// TwinCAT 3 PLC project PLC
// ProgramVersion: 3.1.4023.0
// libraries:
//   Tc2_Standard, * (Beckhoff Automation GmbH)
//   Tc2_System, * (Beckhoff Automation GmbH)
//   Tc3_EventLogger, * (Beckhoff Automation GmbH)
//   Tc3_Module, * (Beckhoff Automation GmbH)
// project tree:
//   GVLs/ GVL.TcGVL
//   / PlcTask.TcTTO
//   POUs/ FB_Alarm.TcPOU, MAIN.TcPOU
// real-time tasks:
//   TASK PlcTask: cycle T#10ms, priority 20, ADS port 350

CONFIGURATION PLC
    RESOURCE PLC ON TwinCAT3
        TASK PlcTask(INTERVAL := T#10ms, PRIORITY := 20);
        PROGRAM MAIN WITH PlcTask : MAIN;
    END_RESOURCE
END_CONFIGURATION

// ---- GVLs/GVL.TcGVL

VAR_GLOBAL

END_VAR

// ---- POUs/MAIN.TcPOU
PROGRAM MAIN
VAR
	// Variables for the FB_TcMessage example
	bInitEvent1 	: BOOL; 
	bInitEvent2 	: BOOL; 
    bSend 			: BOOL; 
	fbMessage 		: FB_TcMessage; 
	
	// Variables for the FB_TcAlarm example
	bAlarmEvent		: BOOL;
	bConfirm		: BOOL;
	bDoSomething	: BOOL := FALSE;
	fbAlarm			: FB_Alarm;

END_VAR

// Message example

IF bInitEvent1 THEN
    bInitEvent1 := FALSE; 
    fbMessage.CreateEx(TC_EVENTS.EventClass.Event1, 0); 
END_IF

IF bInitEvent2 THEN
    bInitEvent2 := FALSE; 
    fbMessage.CreateEx(TC_EVENTS.EventClass.Event2, 0); 
END_IF

IF bSend THEN 
    bSend := FALSE; 
    fbMessage.Send(0); 
END_IF

// Alarm Example
fbAlarm(evtEntry:=TC_Events.EventClass.Event1, bEvt:=bAlarmEvent, bConfirm:=bConfirm);

IF fbAlarm.eConfirmationState = TcEventConfirmationState.WaitForConfirmation THEN
	bDoSomething := TRUE;
ELSE
	bDoSomething := FALSE;
END_IF

END_PROGRAM

// ---- POUs/FB_Alarm.TcPOU
FUNCTION_BLOCK FB_Alarm EXTENDS FB_TcAlarm

VAR_INPUT
	evtEntry	: TcEventEntry;
	bEvt		: BOOL;
	bConfirm	: BOOL;
END_VAR

VAR_OUTPUT
END_VAR

VAR
	bInit  		: BOOL := TRUE;
	bMem		: BOOL;
END_VAR

IF bInit THEN
	SUPER^.CreateEx(evtEntry, TRUE, 0);
	bInit := FALSE;
END_IF

IF bEvt AND NOT bMem AND SUPER^.eConfirmationState <> TcEventConfirmationState.WaitForConfirmation THEN
	SUPER^.Raise(0);
END_IF

IF bMem AND NOT bEvt THEN
	SUPER^.Clear(0, FALSE);
END_IF

IF bConfirm THEN
	SUPER^.Confirm(0);
END_IF

bMem := bEvt;

END_FUNCTION_BLOCK
